TEXTLIST EL1809_M_3
  1 = 'L_rear foot pedal2' | chinese: '左后脚踏开关2' | Chinese: '左后脚踏开关2'
  2 = 'L_rear foot pedal3' | chinese: '左后脚踏开关3' | Chinese: '左后脚踏开关3'
  3 = 'R_rear foot pedal1' | chinese: '右后脚踏开关1' | Chinese: '右后脚踏开关1'
  4 = 'R_rear foot pedal2' | chinese: '右后脚踏开关2' | Chinese: '右后脚踏开关2'
  5 = 'R_rear foot pedal3' | chinese: '右后脚踏开关3' | Chinese: '右后脚踏开关3'
  6 = 'Dul detects  input' | chinese: '单/双roll检测限位input' | Chinese: '单/双roll检测限位input'
  7 = 'Dul detects  output' | chinese: '单/双roll检测限位output' | Chinese: '单/双roll检测限位output'
  8 = 'Chuck up input' | chinese: '卡盘到位检测input' | Chinese: '卡盘到位检测input'
  9 = 'Chuck up output' | chinese: '卡盘到位检测output' | Chinese: '卡盘到位检测output'
  10 = ''
  11 = ''
  12 = ''
  13 = ''
  14 = ''
  15 = ''
  16 = ''
   = ''
END_TEXTLIST

(* stored: Version 1.1.0.1, ProductVersion 3.1.4024.11
   TextList EL1809_M_3: Id {5cfa3280-705b-4ff2-9395-f878dede9527} *)
